# B&R Automation Studio project MotionTestBenchMaster (part 12)

```c
/*============================================================================*/
void mberror_client(tstMBT_SVars* inst, USINT clt)
/*----------------------------------------------------------------------------
  Function:

  History:

  Version | Date        | Author      | Description
  -----------------------------------------------------------------------------
     1.00 | 2010-okt-19 | H.Anderes    | creation
  ============================================================================*/
  {
  /* _LOCAL */
  STRING errstr[5+1];                        /* for status number */
  USINT  msize;                              /* for defensive programming, */
  /* _DYNAMIC */
  /*==========================================================================*/
  msize = sizeof(inst->cltInfo[clt].szMsg) - 1; /* http://www.manpagez.com/man/3/strncat/ */

  memset(inst->cltInfo[clt].szMsg, 0, sizeof(inst->cltInfo[clt].szMsg));
  switch (inst->uiStepCltHandler[clt])
  {
  /*-----------------------------------------------------------------------------
    DEBUG: client_handler state machine: W4_REQUEST
  ------------------------------------------------------------------------------*/
  case enMBTCP_CLT_HANDLER_W4_REQUEST:
    (void)strncat( inst->cltInfo[clt].szMsg,
                   "W4_REQUEST:",
                   msize - strlen(inst->cltInfo[clt].szMsg));
    (void)itoa(inst->stTcpSend[clt].status, (UDINT) &errstr);
    (void)strncat( inst->cltInfo[clt].szMsg,
                   errstr,
                   msize - strlen(inst->cltInfo[clt].szMsg));
    /* verfiy status */
    switch (inst->stTcpRecv[clt].status)
    {
    case ERR_OK:
      (void)strncat(inst->cltInfo[clt].szMsg, " status OK",
                    msize - strlen(inst->cltInfo[clt].szMsg));
      break;
    case ERR_FUB_BUSY:
      (void)strncat(inst->cltInfo[clt].szMsg, " FUB busy, trying again",
                    msize - strlen(inst->cltInfo[clt].szMsg));
      break;
    case tcpERR_NO_DATA:
      (void)strncat(inst->cltInfo[clt].szMsg, " Waiting (NO_DATA)",
                    msize - strlen(inst->cltInfo[clt].szMsg));
      break;
    case tcpERR_INVALID_IDENT:
    case tcpERR_NOT_CONNECTED:
      (void)strncat( inst->cltInfo[clt].szMsg,
                     " INVALID_IDENT, NOT_CONNECTED, disconnecting",
                     msize - strlen(inst->cltInfo[clt].szMsg));
      break;
    case tcpERR_SYSTEM:
      (void)strncat( inst->cltInfo[clt].szMsg,
                     " internal error while receiving",
                     msize - strlen(inst->cltInfo[clt].szMsg));
      /*************************************************************************/
      #ifdef _MBTCP_LOGGER_DEBUG
      ERRxwarning( mbtERR_NOT_CONNECTED,
                   inst->cltInfo[clt].udiIdent,
                   "MBTCP Server: TCP Recv tcpERR_SYSTEM");
      #endif
      /*************************************************************************/
      break;
    /*-------------------------------------------------------------------------*/
    case ERR_FUB_ENABLE_FALSE:
       (void)strncat(inst->cltInfo[clt].szMsg, " FUB not enabled",
                    msize - strlen(inst->cltInfo[clt].szMsg));
       break;
    /*-------------------------------------------------------------------------*/
    case tcpERR_NO_OOBDATA:
    case tcpERR_PARAMETER:
    case tcpERR_INVALID:
    default:
      (void)strncat(inst->cltInfo[clt].szMsg, " unknown error",
                    msize - strlen(inst->cltInfo[clt].szMsg));
      break;
    }
    break;
  /*-----------------------------------------------------------------------------
    DEBUG: client_handler state machine: SEND_RESPONSE
  ------------------------------------------------------------------------------*/
  case enMBTCP_CLT_HANDLER_SEND_RESPONSE:
    (void)strncat( inst->cltInfo[clt].szMsg,
                   "SEND_RESPONSE:",
                   msize - strlen(inst->cltInfo[clt].szMsg));
    (void)itoa(inst->stTcpSend[clt].status, (UDINT) &errstr);
    (void)strncat( inst->cltInfo[clt].szMsg,
                   errstr,
                   msize - strlen(inst->cltInfo[clt].szMsg));
    /* verify status */
    switch (inst->stTcpSend[clt].status)
    {
    case ERR_OK:
      (void)strncat(inst->cltInfo[clt].szMsg, " status OK",
                    msize - strlen(inst->cltInfo[clt].szMsg));
      break;
    case ERR_FUB_BUSY:
      (void)strncat(inst->cltInfo[clt].szMsg, " FUB busy, trying again",
                    msize - strlen(inst->cltInfo[clt].szMsg));
      break;
    case ERR_FUB_ENABLE_FALSE:
      (void)strncat(inst->cltInfo[clt].szMsg, " FUB not enabled",
                    msize - strlen(inst->cltInfo[clt].szMsg));
      break;
    case tcpERR_INVALID_IDENT:
      (void)strncat(inst->cltInfo[clt].szMsg, " ident not available",
                    msize - strlen(inst->cltInfo[clt].szMsg));
      break;
    case tcpERR_PARAMETER:
      (void)strncat(inst->cltInfo[clt].szMsg, " pData not set",
                    msize - strlen(inst->cltInfo[clt].szMsg));
      break;
    case tcpERR_SENTLEN:
      (void)strncat(inst->cltInfo[clt].szMsg,
                    " length of data to send <> specified length",
                    msize - strlen(inst->cltInfo[clt].szMsg));
      break;
    case tcpERR_WOULDBLOCK:
      (void)strncat(inst->cltInfo[clt].szMsg,
                    " data blocked out of socket's send buffer",
                    msize - strlen(inst->cltInfo[clt].szMsg));
      break;
    case tcpERR_NOT_CONNECTED:
      (void)strncat(inst->cltInfo[clt].szMsg,
                    " connection closed by opposite side",
                    msize - strlen(inst->cltInfo[clt].szMsg));
      break;
    case tcpERR_SYSTEM:
      (void)strncat(inst->cltInfo[clt].szMsg, " internal error while sending",
                    msize - strlen(inst->cltInfo[clt].szMsg));
      /************************************************************************/
      #ifdef _MBTCP_LOGGER_DEBUG
      ERRxwarning( mbtERR_NOT_CONNECTED,
                   inst->cltInfo[clt].udiIdent,
                   "MBTCP Server: Tcp Send tcpERR_SYSTEM");
      /************************************************************************/
      #endif
      break;
    default:
      (void)strncat(inst->cltInfo[clt].szMsg, " unknown error",
                    msize - strlen(inst->cltInfo[clt].szMsg));
      break;
    }
    break;
  /*-----------------------------------------------------------------------------
    DEBUG: client_handler state machine: DISCONNECT
  ------------------------------------------------------------------------------*/
  case enMBTCP_CLT_HANDLER_DISCONNECT:
    (void)strncat( inst->cltInfo[clt].szMsg,
                   "DISCONNECT:TCP_CLOSE:",
                   msize - strlen(inst->cltInfo[clt].szMsg));
    (void)itoa(inst->stTcpClose[clt].status, (UDINT) &errstr);
    (void)strncat( inst->cltInfo[clt].szMsg,
                   errstr,
                   msize - strlen(inst->cltInfo[clt].szMsg));
    /* verfiy status */
    switch (inst->stTcpClose[clt].status)
    {
    case ERR_OK:
      (void)strncat(inst->cltInfo[clt].szMsg, " OK. Client connection closed",
                    msize - strlen(inst->cltInfo[clt].szMsg));
      /************************************************************************/
      #ifdef _MBTCP_LOGGER_EVENT
      ERRxwarning( mbtEVENT_CLOSE_CLIENT,
                   inst->stTcpClose[clt].ident,
                   "MBTCP Server: Close Client");
      #endif
      /************************************************************************/
      break;
    case ERR_FUB_BUSY:
      (void)strncat(inst->cltInfo[clt].szMsg, " FUB_BUSY, Still trying...",
                    msize - strlen(inst->cltInfo[clt].szMsg));
      break;
    case tcpERR_INVALID_IDENT:
      (void)strncat(inst->cltInfo[clt].szMsg, " INVALID_IDENT",
                    msize - strlen(inst->cltInfo[clt].szMsg));
      break;
    case ERR_FUB_ENABLE_FALSE:
      (void)strncat(inst->cltInfo[clt].szMsg, " FUB_ENABLE_FALSE",
                    msize - strlen(inst->cltInfo[clt].szMsg));
      break;
    default:
      (void)strncat(inst->cltInfo[clt].szMsg, " unknown error",
                    msize - strlen(inst->cltInfo[clt].szMsg));
      break;
    }
    break;
  }
  /*==========================================================================*/
  } /* mberror */

/******************************************************************************
 * END OF CODE
 ******************************************************************************/
/*
Local Variables:
c-file-style: bsd
c-basic-offset: 2
comment-column: 45
End:
 */
```

#### MBTMaster.h
```c
/*****************************************************************************
 * Copyright:    B&R Industrie-Automation AG
 *
 * Project:      Library MBTCP
 *
 * Target:       B&R-PCC
 *
 * AR-Version:   B 2.01
 *
 * AS-Version:   V 3.0.71.16.SP01
 *
 * Filename:     MBTMaster.h
 *
 * Function:     module-description
 *
 * Dependencies: description of all dependencies
 *
 *****************************************************************************
 * History:
 *
 * Version | Date        | Author      | Description
 * --------------------------------------------------------------------------
 *    1.00 | 2008-Sep-30 | H.Anderes    | creation
 *****************************************************************************/

/*****************************************************************************
 * includes
 *****************************************************************************/
#ifndef MBTMASTER_H_
#define MBTMASTER_H_
/* ansi-c import */
#include <string.h>
/* system import */
#include <bur/plc.h>                         /* IEC data types */
#include <asstring.h>
#include <brsystem.h>
#include <astcp.h>
#include <convert.h>
#include <sys_lib.h>
/* user defined import */
#include "MBTCP.h"

/*#define _MBTCP_LOGGER_DEBUG*/    /* if defined, errors are logged into the logger */
/*#define _MBTCP_LOGGER_EVENT*/    /* if defined, events are logged into the logger */

#ifdef __i386__
#define SWAPUINT        swapUINT
#define SWAPINT         swapINT
#else
#define SWAPUINT
#define SWAPINT
#endif

/*****************************************************************************
 * constants / macros
 *****************************************************************************/
#define NELEMS(array)           (sizeof(array) / sizeof(array[0]))
/* Booleans, switches
 */
enum {
  FALSE                   = 0,
  TRUE                    = 1,
  EXIT_FAILURE            = 1,
  ON                      = 0xFF00,
  OFF                     = 0x0000
};

#define MAX_COILS    2000
#define MAX_REGISTER 127
/*****************************************************************************
 * type definitions
 *****************************************************************************/
/* STEP values
 */
enum {
  INIT                    = 0,
  WAIT_SERVER             = 5,
  OPEN_PORT               = 10,
  IOCTL                   = 15,
  WAIT_CONNECTION         = 20,
  WAIT_REQUEST            = 30,
  SEND_ANSWER             = 40,
  SEND_REQUEST            = 50,
  WAIT_ANSWER             = 60,
  CLOSE_PORT              = 70,
  FATAL_ERROR0            = 240,
  FATAL_ERROR1            = 241,
  FATAL_ERROR2            = 242,
  FATAL_ERROR3            = 243,
  FATAL_ERROR4            = 244,
  FATAL_ERROR5            = 245,
  FATAL_ERROR6            = 246,
  FATAL_ERROR7            = 247,
  FATAL_ERROR8            = 248,
  FATAL_ERROR9            = 249,
  FATAL_ERROR10           = 250,
  FATAL_ERROR             = 251,
  FINAL_ERROR			  = 252,

  DISABLE                 = 65534,
  BUSY                    = 65535
};

/* Modbus function codes
 */
enum {
  READ_COILS                            = 0x01,
  READ_DISCRETE_INPUTS                  = 0x02,
  READ_HOLDING_REGISTERS                = 0x03,
  READ_INPUT_REGISTERS                  = 0x04,
  WRITE_SINGLE_COIL                     = 0x05,
  WRITE_SINGLE_REGISTER                 = 0x06,
  WRITE_MULTIPLE_COILS                  = 0x0F,
  WRITE_MULTIPLE_REGISTERS              = 0x10,
  READ_WRITE_MULTIPLE_REGISTERS         = 0x17
};
/* Modbus protocol exception codes
 */
enum {
  MB_ILLEGAL_FUNCTION                   = 0x01,
  MB_ILLEGAL_DATA_ADDRESS               = 0x02,
  MB_ILLEGAL_DATA_VALUE                 = 0x03,
  MB_SLAVE_DEVICE_FAILURE               = 0x04,
  MB_ACKNOWLEDGE                        = 0x05,
  MB_SLAVE_DEVICE_BUSY                  = 0x06,
  MB_MEMORY_PARITY_ERROR                = 0x08,
  MB_GATEWAY_PATH_UNAVAILABLE           = 0x0A,
  MB_GATEWAY_TARGET_DEV_FAILED_RESPOND  = 0x0B
};
/* Dimensions
 */
enum {
  MBT_SLAVE_PORT        = 502,
  MAX_OPEN_RETRIES      = 3,
  RECV_TIMEOUT_DFLT     = 500,               /* default timeout */
  IPADDR_L              = 18,
  MAX_NBR_REQUESTS      = 5,                 /* was 20 */
  MAX_BUFFER_LEN        = 1200,/*128,*/
  MESS_LEN              = 100,               /* error message length */
};

/* Datatypes */
typedef struct MBTMasterActionParam_typ
{
  USINT usiFCode;
  USINT usiUnit;
  UINT  uiReadAddr;
  UINT  uiReadQty;
  UDINT puiReadVal;
  UINT  uiWriteAddr;
  UINT  uiWriteQty;
  UDINT puiWriteVal;
  UDINT udiTimer;
} MBTMasterActionParam_typ;

typedef struct MBTMasterActionEnable_typ
{
  BOOL bCyclic;
  BOOL bSingle;
} MBTMasterActionEnable_typ;

typedef struct tstMBT_MData
{
  MBTMasterActionEnable_typ actEnable[MAX_NBR_REQUESTS];
  MBTMasterActionParam_typ actParam[MAX_NBR_REQUESTS];
} tstMBT_MData;

typedef struct
{
  BOOL                  bEnable;
  STRING                slvIPAddr[IPADDR_L];
  UINT                  uiPort;
  UINT                  uiRecvTimeout;
  UDINT                 udiCycleTime;
  tstMBT_MData*         pData;
  UINT                  uiStep;
  TcpOpen_typ           stTcpOpen;
  TcpIoctl_typ          stTcpIoctl;
  TcpClient_typ         stTcpClient;
  TcpSend_typ           stTcpSend;
  TcpRecv_typ           stTcpRecv;
  TcpClose_typ          stTcpClose;
  USINT                 usiLastReq;
  UDINT                 udiRecvTimer;
  UDINT                 udiSendTimer[MAX_NBR_REQUESTS];
  USINT                 usiSendBuf[MAX_BUFFER_LEN];
  USINT                 usiRecvBuf[MAX_BUFFER_LEN];
  BOOL                  bRecvOK;
  UINT                  uiStatus;
  UINT                  uiTxID;
  UDINT                 udiWrongMsg;
  STRING                szMsg[MESS_LEN];
  tcpLINGER_typ         mLinger;
  USINT                 usiOpenRetries;
  USINT                 usiSendCnt;
} tstMBT_MVars;

/*****************************************************************************
 * functions protoytpes
 ****************************************************************************/
void  fMBTMStates(tstMBT_MVars* inst);
UINT create_request_to_server(tstMBT_MVars*   inst,
                               tstMBT_MData*   config,
                               USINT           usiOp,
                               USINT*          usiSendBuf,
                               UINT            uiTxID);
USINT analyze_answer_from_server(tstMBT_MVars* inst,
                                 tstMBT_MData* config,
                                 USINT         usiOp,
                                 USINT*        usiRecvBuf,
                                 UINT          uiTxID);

/****************************************************************************
 * END OF CODE
 ****************************************************************************/
/*
Local Variables:
c-file-style: bsd
c-basic-offset: 2
comment-column: 45
End:
 */
#endif /* MBTMASTER_H_ */
```

#### MBTMaster.c
```c
/******************************************************************************
 * Copyright:    B&R Industrie-Automation AG
 *
 * Project:      Library MBTCP
 *
 * Target:       B&R-PCC
 *
 * AR-Version:   B 2.01
 *
 * AS-Version:   V 3.0.71.16.SP01
 *
 * Filename:     MBTMaster.c
 *
 * Function:     module-description
 *
 * Dependencies: description of all dependencies
 *
 ******************************************************************************
 * History:
 *
 * Version | Date        | Author      | Description
 * ----------------------------------------------------------------------------
 *    1.00 | 2008-Sep-30 | H.Anderes   | creation
 *    2.00 | 2010-okt-04 | H.Anderes   | refactory
 *****************************************************************************/

/******************************************************************************
 * includes
 *****************************************************************************/
/* ansi-c import */
/* system import */
/* user defined import */
#include "MBTMaster.h"

/******************************************************************************
 * functions
 ******************************************************************************/
/*============================================================================*/
void fMBTMStates(tstMBT_MVars* inst)
/*----------------------------------------------------------------------------
  Function:

  History:

  Version | Date        | Author      | Description
  ----------------------------------------------------------------------------
  1.00    | 2008-sep-30 | H.Anderes    | creation
  2.00    | 2010-okt-04 | H.Anderes   | refactory
  ============================================================================*/
{
  /* _LOCAL */
  UINT uiFatalErrNum;
  USINT i, usiOp;                            /* usiOp: number of operations */
  USINT recv_status;
  /* _DYNAMIC */
  /*==========================================================================*/
  /* check if a null pointer is passed to the fub */
  if (inst == NULL)
  {
    return;
  }
  /*--------------------------------------------------------------------------------
    state machine : Modbus TCP Master
  ---------------------------------------------------------------------------------*/
  switch(inst->uiStep)
  {
  /*-----------------------------------------------------------------------------
    INIT: initialize TcpSend and TCPRecv
  ------------------------------------------------------------------------------*/
  case INIT:
    inst->stTcpSend.pData   = (UDINT)inst->usiSendBuf;
    inst->stTcpRecv.pData   = (UDINT)inst->usiRecvBuf;
    inst->stTcpRecv.datamax = MAX_BUFFER_LEN;
    inst->uiStep            = DISABLE;
    /* FALL THROUGH */
  /*-----------------------------------------------------------------------------
    DISBALE: waits until the fub is enabled
  ------------------------------------------------------------------------------*/
  case DISABLE:
    if(inst->bEnable)
    {
      inst->uiStep = OPEN_PORT;
    }
    break;
  /*-----------------------------------------------------------------------------
    OPEN: opens a TCP - socket
  ------------------------------------------------------------------------------*/
  case OPEN_PORT:
    inst->stTcpOpen.enable = 1;
    inst->stTcpOpen.port   = 0;
    /* call TcpOpen() */
    TcpOpen(&inst->stTcpOpen);
    /* verfiy status */
    switch (inst->stTcpOpen.status)
    {
    /*-------------------------------------------------------------------------*/
    case ERR_OK:
      inst->stTcpClient.enable     = 1;
      inst->stTcpClient.ident      = inst->stTcpOpen.ident;
      inst->stTcpClient.pServer    = (UDINT)inst->slvIPAddr;
      inst->stTcpClient.portserv   = inst->uiPort;
      inst->stTcpSend.ident        = inst->stTcpOpen.ident;
      inst->stTcpRecv.ident        = inst->stTcpOpen.ident;
      inst->uiStep                 = IOCTL;
      /************************************************************************/
      #ifdef _MBTCP_LOGGER_EVENT
	     ERRxwarning( mbtEVENT_OPEN_PORT,
                   inst->stTcpOpen.ident,
                   "MBTCP Client: Open Port");
      #endif
      /************************************************************************/
      break;
    /*-------------------------------------------------------------------------*/
    case ERR_FUB_BUSY:
      /* do nothing */
      break;
    /*-------------------------------------------------------------------------*/
    case tcpERR_NOMORE_IDENTS:
    case tcpERR_ALREADY_EXIST:
    case tcpERR_SOCKET_CREATE:
    case tcpERR_SOCKET_BIND:
    case tcpERR_INTERFACE:
    case tcpERR_SYSTEM:
    case ERR_FUB_ENABLE_FALSE:
    default:
      inst->uiStatus = inst->stTcpOpen.status;
      inst->uiStep   = FATAL_ERROR0;
      break;
    }
    break;
  /*-----------------------------------------------------------------------------
    IOCTRL: configuration of the TCP - connection
  ------------------------------------------------------------------------------*/
  case IOCTL:
    /* set linger that the connection is not abort immediately */
    inst->mLinger.lOnOff     = 0;
    inst->mLinger.lLinger    = 0;
     /* initialize fub */
    inst->stTcpIoctl.enable 	= 1;
    inst->stTcpIoctl.ident	  = inst->stTcpOpen.ident;
    inst->stTcpIoctl.ioctl 	 = tcpSO_LINGER_SET;
    inst->stTcpIoctl.pData	  = (UDINT)&inst->mLinger;
    inst->stTcpIoctl.datalen	= sizeof(tcpLINGER_typ);
    /* call  TcpIoctl()n */
    TcpIoctl(&inst->stTcpIoctl);
    /* verify status */
    switch (inst->stTcpIoctl.status)
    {
    /*-------------------------------------------------------------------------*/
    case ERR_OK:
      inst->usiOpenRetries = 0;      /* we reset prior to next step */
      inst->uiStep         = WAIT_CONNECTION;
      break;
    /*-------------------------------------------------------------------------*/
    case ERR_FUB_BUSY:
      inst->uiStep = IOCTL;
      break;
    /*-------------------------------------------------------------------------*/
    case tcpERR_INVALID_IDENT:
      inst->uiStatus = inst->stTcpIoctl.status;
      if (inst->usiOpenRetries < MAX_OPEN_RETRIES)
      {
        inst->uiStep = OPEN_PORT;
        inst->usiOpenRetries++;
        /************************************************************************/
        #ifdef _MBTCP_LOGGER_DEBUG
		      ERRxwarning( mbtERR_OPEN_RETRIES_IOC,
                     inst->stTcpOpen.ident,
                     "MBTCP Client: OPEN Retries IOCTL");
        #endif
        /************************************************************************/
      }
      else
      {
        inst->uiStep = FATAL_ERROR1;
      }
      break;
    /*-------------------------------------------------------------------------*/
    case tcpERR_PARAMETER:
      inst->uiStatus = inst->stTcpIoctl.status;
      inst->uiStep   = CLOSE_PORT;
      break;
    /*-------------------------------------------------------------------------*/
    case tcpERR_INVALID_IOCTL:
    case ERR_FUB_ENABLE_FALSE:
    default:
      inst->uiStatus = inst->stTcpIoctl.status;
      inst->uiStep   = FATAL_ERROR2;
      break;
    }
    break;
  /*-----------------------------------------------------------------------------
    WAIT: waits until a connection to a TCP Server is acc
  ------------------------------------------------------------------------------*/
  case WAIT_CONNECTION:
    inst->stTcpClient.enable = 1;
    /* call TcpClient() */
    TcpClient(&inst->stTcpClient);
    /* verify status */
    switch (inst->stTcpClient.status)
    {
    /*-------------------------------------------------------------------------*/
    case ERR_OK:
      inst->uiStep = SEND_REQUEST;
      break;
    /*-------------------------------------------------------------------------*/
    case ERR_FUB_BUSY:
      /* do nothing */
	     strcpy( inst->szMsg,
              "WAIT_CONNECTION:TcpClient: Wait Connection");
      break;
    /*-------------------------------------------------------------------------*/
    case tcpERR_INVALID:
   	  inst->uiStep = CLOSE_PORT;
      /*************************************************************************/
      #ifdef _MBTCP_LOGGER_DEBUG
   	  ERRxwarning( tcpERR_INVALID,
                   inst->stTcpClient.ident,
                   "MBTCP Client: Wait connecction; Invalid ");
      #endif
      /*************************************************************************/
      break;
    /*-------------------------------------------------------------------------*/
    case tcpERR_ALREADY_CONNECTED:
      inst->uiStep = CLOSE_PORT;
      /*************************************************************************/
      #ifdef _MBTCP_LOGGER_DEBUG
	     ERRxwarning( tcpERR_ALREADY_CONNECTED,
                             inst->stTcpClient.ident,
                             "MBTCP Client: Wait connecction; Already connected");
      #endif
      /*************************************************************************/
      break;
    /*-------------------------------------------------------------------------*/
    case tcpERR_SYSTEM:
    case ERR_FUB_ENABLE_FALSE:
    default:
      inst->uiStep = FATAL_ERROR3;
      break;
    }
    break;
  /*-----------------------------------------------------------------------------
    CREATE: creates the request
  ------------------------------------------------------------------------------*/
  case SEND_REQUEST:
    if (inst->bEnable)
    {
      inst->bRecvOK = FALSE;
      /* cycle through list of Modbus operations for MAX_NBR_REQUESTS times */
      for (i = inst->usiLastReq + 1;
           i < (MAX_NBR_REQUESTS + inst->usiLastReq + 1);
           i++)
      {
        usiOp = i % MAX_NBR_REQUESTS;
        if ((*(inst->pData)).actEnable[usiOp].bSingle)
        {
          inst->udiSendTimer[usiOp] =
            (*(inst->pData)).actParam[usiOp].udiTimer;
        }
        if ( (((*(inst->pData)).actEnable[usiOp].bCyclic)
              || ((*(inst->pData)).actEnable[usiOp].bSingle)))
        {
          if (inst->udiSendTimer[usiOp]
              >= (*(inst->pData)).actParam[usiOp].udiTimer)
          {
            inst->usiLastReq = usiOp;
            inst->uiStep = SEND_REQUEST + 1;
            inst->uiTxID++;
            inst->stTcpSend.datalen =
                create_request_to_server((tstMBT_MVars*)(inst),
                                       (tstMBT_MData*)(inst->pData),
                                       usiOp,
                                       inst->usiSendBuf,
                                       inst->uiTxID);
            inst->udiSendTimer[usiOp] = 0;
            break;
          }
          else
          {
            inst->udiSendTimer[usiOp] += inst->udiCycleTime;
          }
        }
        else
        {
          inst->udiSendTimer[usiOp]
            = (*(inst->pData)).actParam[usiOp].udiTimer;
        }
      }
    }
    else
    {
      inst->uiStep = CLOSE_PORT;
    }
    break;
  /*-----------------------------------------------------------------------------
    SEND: sends the created request to the server/slave
  ------------------------------------------------------------------------------*/
  case SEND_REQUEST + 1:
    if (inst->bEnable)
    {
      inst->stTcpSend.enable = 1;
      /* call TcpSend() */
      TcpSend(&inst->stTcpSend);
      /* verfiy status */
      switch (inst->stTcpSend.status)
      {
      /*-------------------------------------------------------------------------*/
      case ERR_OK:
        inst->usiSendCnt   = 0;
        inst->udiRecvTimer = 0;
        inst->uiStep       = WAIT_ANSWER;
        break;
      /*-------------------------------------------------------------------------*/
      case ERR_FUB_BUSY:
	       /* do nothing */
		      strcpy( inst->szMsg,
                "SEND_REQUEST + 1:TcpSend: ERR_FUB_BUSY");
	  	    break;
      /*-------------------------------------------------------------------------*/
      case tcpERR_WOULDBLOCK:
         /* send again */
         /************************************************************************/
         #ifdef _MBTCP_LOGGER_DEBUG
  	      ERRxwarning( tcpERR_WOULDBLOCK,
                      inst->stTcpClient.ident,
                      "MBTCP Client: Wouldblock");
         #endif
         /***********************************************************************/
   	   	break;
      /*-------------------------------------------------------------------------*/
      case tcpERR_SENTLEN:
        /* send length not ok. send again */
        /************************************************************************/
        #ifdef _MBTCP_LOGGER_DEBUG
        ERRxwarning( tcpERR_SENTLEN,
                     inst->stTcpClient.ident,
                     "MBTCP Client: Send lenght not Ok");
        #endif
        /************************************************************************/
        break;
      /*------------------------------------------------------------------------*/
      case tcpERR_NOT_CONNECTED:
        inst->uiStep = CLOSE_PORT;
        /************************************************************************/
        #ifdef _MBTCP_LOGGER_DEBUG
		      ERRxwarning( tcpERR_NOT_CONNECTED,
                     inst->stTcpClient.ident,
                     "MBTCP Client: Not connected");
        #endif
        /************************************************************************/
        break;
      /*-------------------------------------------------------------------------*/
      case tcpERR_INVALID_IDENT:
      case tcpERR_PARAMETER:
      case tcpERR_SYSTEM:
      default:
        inst->uiStep = FATAL_ERROR4;
        break;
      }
    }
    else
    {
      inst->uiStep = CLOSE_PORT;
    }
    break;
  /*-----------------------------------------------------------------------------
    WAIT: waits until a response is received or a timeout occured
  ------------------------------------------------------------------------------*/
  case WAIT_ANSWER:
    if (inst->bEnable)
    {
      inst->udiRecvTimer += inst->udiCycleTime;
      if (inst->udiRecvTimer >= inst->uiRecvTimeout)
      {
        /* send again after timeout */
        inst->uiStep = SEND_REQUEST;
        /************************************************************************/
        #ifdef _MBTCP_LOGGER_DEBUG
		      ERRxwarning( mbtERR_TIMEOUT,
                     inst->stTcpClient.ident,
                     "MBTCP Client: Receive Timeout");
        #endif
        /************************************************************************/
        break;
      }
      inst->stTcpRecv.enable = 1;
      /* call TcpRecv() */
      TcpRecv(&(inst->stTcpRecv));
      /* verfiy status */
      switch (inst->stTcpRecv.status)
      {
      /*-------------------------------------------------------------------------*/
      case ERR_OK:
        if (inst->stTcpRecv.recvlen > 8)
        {
          recv_status =
            analyze_answer_from_server((tstMBT_MVars*)(inst),
                                       (tstMBT_MData*)(inst->pData),
                                       inst->usiLastReq,
                                       inst->usiRecvBuf,
                                       inst->uiTxID);
        }
        else
        {
          recv_status = 1;
        }
        if(recv_status)
		      {
           inst->udiWrongMsg++;
           /**********************************************************************/
           #ifdef _MBTCP_LOGGER_DEBUG
 		        ERRxwarning( mbtERR_RESPONSE,
                        inst->stTcpRecv.ident,
                        "MBTCP Client: Response not Ok");
           #endif
           /**********************************************************************/

        }
        else
        {
          (*(inst->pData)).actEnable[inst->usiLastReq].bSingle = 0;
        }
        inst->uiStep = SEND_REQUEST;
        break;
      /*-------------------------------------------------------------------------*/
      case ERR_FUB_BUSY:
      case ERR_FUB_ENABLE_FALSE:
      case tcpERR_NO_DATA:
        /* do nothing */
		      strcpy(inst->szMsg, "WAIT_ANSWER:TcpClient: tcpERR_NO_DATA");
        break;
      /*-------------------------------------------------------------------------*/
      case tcpERR_NOT_CONNECTED:
        inst->uiStep = SEND_REQUEST;
		      strcpy(inst->szMsg, "WAIT_ANSWER:TcpClient: tcpERR_NOT_CONNECTED");
        break;
      /*-------------------------------------------------------------------------*/
      case tcpERR_INVALID_IDENT:
      case tcpERR_PARAMETER:
      case tcpERR_INVALID:
      case tcpERR_NO_OOBDATA:
      case tcpERR_SYSTEM:
      default:
        inst->uiStep = FATAL_ERROR5;
        break;
      }
    }
    else
    {
      inst->uiStep = CLOSE_PORT;
    }
    break;
  /*-----------------------------------------------------------------------------
    CLOSE: closes the TCP - Socket
  ------------------------------------------------------------------------------*/
  case CLOSE_PORT:
    inst->stTcpClose.enable = 1;
    inst->stTcpClose.ident  = inst->stTcpOpen.ident;
    /*
      inst->stTcpClose.how    = tcpSHUT_RD | tcpSHUT_WR;
    */
    inst->stTcpClose.how    = 0;
    /* call TcpClose() */
    TcpClose(&inst->stTcpClose);
    /* verfiy status */
    switch (inst->stTcpClose.status)
    {
    /*-------------------------------------------------------------------------*/
    case ERR_OK:
      inst->uiStep = DISABLE;
      /*************************************************************************/
      #ifdef _MBTCP_LOGGER_DEBUG
	     ERRxwarning( mbtEVENT_CLOSE_PORT,
                   inst->stTcpClose.ident,
                   "MBTCP Client: Close Port");
      #endif
      /*************************************************************************/
      break;
    /*-------------------------------------------------------------------------*/
    case ERR_FUB_BUSY:
      /* do nothing */
      break;
    /*-------------------------------------------------------------------------*/
    case tcpERR_INVALID_IDENT:
      inst->uiStep = WAIT_CONNECTION;
      break;
    /*-------------------------------------------------------------------------*/
    case ERR_FUB_ENABLE_FALSE:
    default:
      inst->uiStep = FATAL_ERROR6;
      break;
    }
    break;
  /*-----------------------------------------------------------------------------
    FATAL ERROR: a fatal error occured
  ------------------------------------------------------------------------------*/
  case FATAL_ERROR0:
  case FATAL_ERROR1:
  case FATAL_ERROR2:
  case FATAL_ERROR3:
  case FATAL_ERROR4:
  case FATAL_ERROR5:
  case FATAL_ERROR6:
  default:
   /* vefiy in which state the fatal error occured */
  	switch(inst->uiStep)
	  {
	  case FATAL_ERROR0: uiFatalErrNum = 0; break;
  	case FATAL_ERROR1: uiFatalErrNum = 1; break;
  	case FATAL_ERROR2: uiFatalErrNum = 2; break;
  	case FATAL_ERROR3: uiFatalErrNum = 3; break;
  	case FATAL_ERROR4: uiFatalErrNum = 4; break;
  	case FATAL_ERROR5: uiFatalErrNum = 5; break;
  	case FATAL_ERROR6: uiFatalErrNum = 6; break;
	  default:
		   uiFatalErrNum = 7; break;
	  }
	   /*************************************************************************/
    #ifdef _MBTCP_LOGGER_DEBUG
   	ERRxwarning( mbtERR_FATAL_ERROR,
                 uiFatalErrNum,
                 "MBTCP Client: FATAL ERROR State Machine");
    #endif
    /*************************************************************************/
   	inst->uiStep = FINAL_ERROR;
    break;

  case FINAL_ERROR:
  	/*Do nothing until Reboot RPS*/
  	break;
  }
}

/*============================================================================*/
UINT create_request_to_server(tstMBT_MVars* inst,
                               tstMBT_MData* config,
                               USINT         usiOp,
                               USINT*        usiSendBuf,
                               UINT          uiTxID)
/*----------------------------------------------------------------------------
  Function:

  History:

  Version | Date        | Author      | Description
  ----------------------------------------------------------------------------
     1.00 | 2008-sep-30 | H.Anderes    | creation
  ============================================================================*/
{
  UINT  uint_var, data_len, i;
  INT  int_var;
  UINT  value;
  UINT  val;
 /*==========================================================================*/
  data_len = 0;

  memset(usiSendBuf, 0, MAX_BUFFER_LEN);
  /* Transaction id: 2 bytes */
  uint_var = SWAPUINT(uiTxID);
  memmove(&usiSendBuf[0], &uint_var, sizeof(uint_var));
  /* Protocol id: 2 bytes */
  uint_var = 0;
  memmove(&usiSendBuf[2], &uint_var, sizeof(uint_var));
  /* Length: 2 bytes */
  /* Unit: 1 byte */
  usiSendBuf[6] = (*config).actParam[usiOp].usiUnit;

  switch((*config).actParam[usiOp].usiFCode)
  {
  /*-------------------------------------------------------------------------
      READ: read coils
  --------------------------------------------------------------------------*/
  case READ_COILS:
    /* Function code: 1 byte */
    usiSendBuf[7] = READ_COILS;
    /* Starting address: 2 bytes */
    uint_var = SWAPUINT((*config).actParam[usiOp].uiReadAddr);
    memmove(&usiSendBuf[8], &uint_var, sizeof(uint_var));
    /* Coils number: 2 bytes */
    uint_var = SWAPUINT((*config).actParam[usiOp].uiReadQty);
    memmove(&usiSendBuf[10], &uint_var, sizeof(uint_var));
    /* Data len */
    data_len = 6;
    inst->bRecvOK = FALSE;
    break;
  /*-------------------------------------------------------------------------
      READ: read discrete inputs
  --------------------------------------------------------------------------*/
  case READ_DISCRETE_INPUTS:
    /* Function code: 1 byte */
    usiSendBuf[7] = READ_DISCRETE_INPUTS;
    /* Starting address: 2 bytes */
    uint_var = SWAPUINT((*config).actParam[usiOp].uiReadAddr);
    memmove(&usiSendBuf[8], &uint_var, sizeof(uint_var));
    /* Inputs number: 2 bytes */
    uint_var = SWAPUINT((*config).actParam[usiOp].uiReadQty);
    memmove(&usiSendBuf[10], &uint_var, sizeof(uint_var));
    /* Data len */
    data_len = 6;
    inst->bRecvOK = FALSE;
    break;
  /*-------------------------------------------------------------------------
      READ: read holding registers
  --------------------------------------------------------------------------*/
  case READ_HOLDING_REGISTERS:
    /* Function code: 1 byte */
    usiSendBuf[7] = READ_HOLDING_REGISTERS;
    /* Starting address: 2 bytes */
    uint_var = SWAPUINT((*config).actParam[usiOp].uiReadAddr);
    memmove(&usiSendBuf[8], &uint_var, sizeof(uint_var));
    /* Holding registers number: 2 bytes */
    uint_var = SWAPUINT((*config).actParam[usiOp].uiReadQty);
    memmove(&usiSendBuf[10], &uint_var, sizeof(uint_var));
    /* Data len */
    data_len = 6;
    inst->bRecvOK = FALSE;
    break;
  /*-------------------------------------------------------------------------
      READ: read input registers
  --------------------------------------------------------------------------*/
  case READ_INPUT_REGISTERS:
    /* Function code: 1 byte */
    usiSendBuf[7] = READ_INPUT_REGISTERS;
    /* Starting address: 2 bytes */
    uint_var = SWAPUINT((*config).actParam[usiOp].uiReadAddr);
    memmove(&usiSendBuf[8], &uint_var, sizeof(uint_var));
    /* Input registers number: 2 bytes */
    uint_var = SWAPUINT((*config).actParam[usiOp].uiReadQty);
    memmove(&usiSendBuf[10], &uint_var, sizeof(uint_var));
    /* Data len */
    data_len = 6;
    inst->bRecvOK = FALSE;
    break;
  /*-------------------------------------------------------------------------
      WRITE: write single coil
  --------------------------------------------------------------------------*/
  case WRITE_SINGLE_COIL:
    /* Function code: 1 byte */
    usiSendBuf[7] = WRITE_SINGLE_COIL;
    /* Starting address: 2 bytes */
    uint_var = SWAPUINT((*config).actParam[usiOp].uiWriteAddr);
    memmove(&usiSendBuf[8], &uint_var, sizeof(uint_var));
    /* Value: 2 bytes */
    memmove(&val, (UINT *)((*config).actParam[usiOp].puiWriteVal), sizeof(UINT));
    if ((BOOL)(val))
      value = ON;
    else
      value = OFF;
    int_var = SWAPUINT(value);
    memmove(&usiSendBuf[10], &int_var, sizeof(int_var));
    /* Data len */
    data_len = 6;
    inst->bRecvOK = FALSE;
    break;
  /*-------------------------------------------------------------------------
      WRITE: write single register
  --------------------------------------------------------------------------*/
  case WRITE_SINGLE_REGISTER:
    /* Function code: 1 byte */
    usiSendBuf[7] = WRITE_SINGLE_REGISTER;
    /* Starting address: 2 bytes */
    uint_var = SWAPUINT((*config).actParam[usiOp].uiWriteAddr);
    memmove(&usiSendBuf[8], &uint_var, sizeof(uint_var));
    /* Value: 2 bytes */
    memmove(&val, (UINT *)(*config).actParam[usiOp].puiWriteVal, sizeof(UINT));
    value = (UINT)(val);
    uint_var = SWAPUINT(value);
    memmove(&usiSendBuf[10], &uint_var, sizeof(uint_var));
    /* Data len */
    data_len = 6;
    inst->bRecvOK = FALSE;
    break;
  /*-------------------------------------------------------------------------
      WRITE: write multiple coils
  --------------------------------------------------------------------------*/
  case WRITE_MULTIPLE_COILS:
    /* Function code: 1 byte */
    usiSendBuf[7] = WRITE_MULTIPLE_COILS;
    /* Starting address: 2 bytes */
    uint_var = SWAPUINT((*config).actParam[usiOp].uiWriteAddr);
    memmove(&usiSendBuf[8], &uint_var, sizeof(uint_var));
    /* Quantity: 2 bytes */
    uint_var = SWAPUINT((*config).actParam[usiOp].uiWriteQty);
    memmove(&usiSendBuf[10], &uint_var, sizeof(uint_var));
    /* Byte count: 1 byte */
    /* Number of usiSendBuf bytes needed to contain data */
    /* less than 8 binary digits: 1 byte */
    if ( (*config).actParam[usiOp].uiWriteQty % 8)
      usiSendBuf[12] = ((*config).actParam[usiOp].uiWriteQty / 8) + 1;
    else      /* more than 8 binary digits: quantity / 8 bytes */
      usiSendBuf[12] = (*config).actParam[usiOp].uiWriteQty / 8;
    /* Coil value: x byte */
    for (i = 0; i < (*config).actParam[usiOp].uiWriteQty; i++)
    {
      memmove(&val,
              (UINT *)((*config).actParam[usiOp].puiWriteVal  +  i * sizeof(UINT)),
              sizeof(UINT));
      if ((BOOL)(val))
        usiSendBuf[13 + (i/8)]
          = usiSendBuf[13 + (i/8)] | (USINT)(0x01 << (i%8));
      else
        usiSendBuf[13 + (i/8)]
          = usiSendBuf[13 + (i/8)] & (USINT)~(0x01 << (i%8));
    }
    /* Data len */
    data_len = 7 + usiSendBuf[12];
    inst->bRecvOK = FALSE;
    break;
  /*-------------------------------------------------------------------------
      WRITE: write multiple registers
  --------------------------------------------------------------------------*/
  case WRITE_MULTIPLE_REGISTERS:
    /* Function code: 1 byte */
    usiSendBuf[7] = WRITE_MULTIPLE_REGISTERS;
    /* Starting address: 2 bytes */
    uint_var = SWAPUINT((*config).actParam[usiOp].uiWriteAddr);
    memmove(&usiSendBuf[8], &uint_var, sizeof(uint_var));
    /* Quantity: 2 bytes */
    uint_var = SWAPUINT((*config).actParam[usiOp].uiWriteQty);
    memmove(&usiSendBuf[10], &uint_var, sizeof(uint_var));
    /* Byte count: 1 byte */
    usiSendBuf[12] = (*config).actParam[usiOp].uiWriteQty * 2;
    /* Coil value: x byte */
    for(i = 0; i < (*config).actParam[usiOp].uiWriteQty; i++)
    {
      value = ((INT*)((*config).actParam[usiOp].puiWriteVal))[i];
      int_var = SWAPINT(value);
      memmove(&usiSendBuf[13 + (i*2)], &int_var, sizeof(int_var));
    }
    /* Data len */
    data_len = 7 + usiSendBuf[12];
    inst->bRecvOK = FALSE;
    break;
  /*-------------------------------------------------------------------------
     READ WRITE:read  write multiple registers
  --------------------------------------------------------------------------*/
  case READ_WRITE_MULTIPLE_REGISTERS:
    /* Function code: 1 byte */
    usiSendBuf[7] = READ_WRITE_MULTIPLE_REGISTERS;
    /* Read starting address: 2 bytes */
    uint_var = SWAPUINT((*config).actParam[usiOp].uiReadAddr);
    memmove(&usiSendBuf[8], &uint_var, sizeof(uint_var));
    /* Read quantity: 2 bytes */
    uint_var = SWAPUINT((*config).actParam[usiOp].uiReadQty);
    memmove(&usiSendBuf[10], &uint_var, sizeof(uint_var));
    /* Write starting address: 2 bytes */
    uint_var = SWAPUINT((*config).actParam[usiOp].uiWriteAddr);
    memmove(&usiSendBuf[12], &uint_var, sizeof(uint_var));
    /* write quantity: 2 bytes */
    uint_var = SWAPUINT((*config).actParam[usiOp].uiWriteQty);
    memmove(&usiSendBuf[14], &uint_var, sizeof(uint_var));
    /* Byte count: 1 byte */
    usiSendBuf[16] = (*config).actParam[usiOp].uiWriteQty * 2;
    /* Coil value: x byte */
    for(i = 0; i < (*config).actParam[usiOp].uiWriteQty; i++)
    {
      value = ((INT*)((*config).actParam[usiOp].puiWriteVal))[i];
      int_var = SWAPINT(value);
      memmove(&usiSendBuf[17 + (i*2)], &int_var, sizeof(int_var));
    }
    /* Data len */
    data_len = 11 + usiSendBuf[16];
    inst->bRecvOK = FALSE;
    break;
  default:
    break;
  }
  /* Length: 2 bytes */
  uint_var = SWAPUINT(data_len);
  memmove(&usiSendBuf[4], &uint_var, sizeof(uint_var));

  return (6 + data_len);
}

 /*==========================================================================*/
USINT analyze_answer_from_server(tstMBT_MVars* inst,
                                 tstMBT_MData* config,
                                 USINT         usiOp,
                                 USINT*        usiRecvBuf,
                                 UINT          uiTxID)
/*----------------------------------------------------------------------------
  Function:

  History:

  Version | Date        | Author      | Description
  ----------------------------------------------------------------------------
     1.00 | 2008-sep-30 | H.Anderes   | creation
     2.00 | 2010-okt-04 | H.Anderes   | refactory
  ============================================================================*/
{
  INT   int_var;
  UINT  uint_var, recv_tr_id, protocol_id, length, uiQty,i;
  USINT unit, function_code;
  UINT  coil_val, di_val;         /* was UDINT */
  /*==========================================================================*/

  coil_val = 0;
  di_val   = 0;
  /* (byte 0,1)  transition is */
  memmove(&uint_var, &(usiRecvBuf[0]), sizeof(uint_var));
  recv_tr_id = SWAPUINT(uint_var);
  /* (byte 2,3)  protocol id */
  memmove(&uint_var, &(usiRecvBuf[2]), sizeof(uint_var));
  protocol_id = SWAPUINT(uint_var);
  /* (byte 4,5)  length */
  memmove(&uint_var, &(usiRecvBuf[4]), sizeof(uint_var));
  length = SWAPUINT(uint_var);
  /* (byte 4,5)  length */
  unit = usiRecvBuf[6];
  /* (byte 7 ) function code */
  function_code = usiRecvBuf[7];

  if (    (recv_tr_id == uiTxID)
       && (protocol_id == 0)
       && (length > 0)
       && (function_code  < 0x80) )
  {

    switch(function_code)
    {
    /*-------------------------------------------------------------------------
      READ: read coils
    --------------------------------------------------------------------------*/
    case READ_COILS:
      /* Quantity: 1 byte */
      uiQty = usiRecvBuf[8];
      if (uiQty > MAX_COILS)
      {
        uiQty = MAX_COILS;
      }
      /* Coil value: x bytes */
      /* uiQty is number of bytes received */
      for (i = 0;(i < uiQty*8) && (i < (*config).actParam[usiOp].uiReadQty); i++) {
        coil_val = (UINT)(usiRecvBuf[9 + (i/8)] & (USINT)(0x01 << (i%8)));
        if ((BOOL)(coil_val))
          ((INT*)((*config).actParam[usiOp].puiReadVal))[i] = 1;
        else
          ((INT*)((*config).actParam[usiOp].puiReadVal))[i] = 0;
      }
      inst->bRecvOK = TRUE;
      break;
    /*-------------------------------------------------------------------------
      READ: read discrete inputs
    --------------------------------------------------------------------------*/
    case READ_DISCRETE_INPUTS:
      /* Quantity: 1 byte */
      uiQty = usiRecvBuf[8];
      if (uiQty > MAX_COILS)
      {
        uiQty = MAX_COILS;
      }
      /* Coil value: x byte */
      /* quantity is number of bytes received */
      for(i = 0; (i < uiQty*8) && (i < (*config).actParam[usiOp].uiReadQty); i++) {
        di_val = (UINT)(usiRecvBuf[9 + (i/8)] & (USINT)(0x01 << (i%8)));
         if ((BOOL)(di_val))
           ((INT*)((*config).actParam[usiOp].puiReadVal))[i] = 1;
         else
           ((INT*)((*config).actParam[usiOp].puiReadVal))[i] = 0;
      }
      inst->bRecvOK = TRUE;
      break;
    /*-------------------------------------------------------------------------
      READ: read hoding registers
    --------------------------------------------------------------------------*/
    case READ_HOLDING_REGISTERS:
      /* Quantity: 1 byte */
       uiQty = usiRecvBuf[8] / 2;
       if (uiQty > MAX_REGISTER)
       {
         uiQty = MAX_REGISTER;
       }
      /* Coil value: x byte */
      for(i = 0; i < uiQty; i++) {
        memmove(&int_var, &usiRecvBuf[9 + (i*2)], sizeof(int_var));
        ((INT*)((*config).actParam[usiOp].puiReadVal))[i] = SWAPINT(int_var);
      }
      inst->bRecvOK = TRUE;
      break;
    /*-------------------------------------------------------------------------
      READ: read input registers
    --------------------------------------------------------------------------*/
    case READ_INPUT_REGISTERS:
      /* Quantity: 1 byte */
      uiQty = usiRecvBuf[8] / 2;
      if (uiQty > MAX_REGISTER)
      {
        uiQty = MAX_REGISTER;
      }
      /* Coil value: x byte */
      for(i = 0; i < uiQty; i++) {
        memmove(&int_var, &usiRecvBuf[9 + (i*2)], sizeof(int_var));
        ((INT*)((*config).actParam[usiOp].puiReadVal))[i] = SWAPINT(int_var);
      }
      inst->bRecvOK = TRUE;
      break;
    /*-------------------------------------------------------------------------
      READ: read write multiple registers
    --------------------------------------------------------------------------*/
    case READ_WRITE_MULTIPLE_REGISTERS:
      /* Quantity: 1 byte */
      uiQty = usiRecvBuf[8] / 2;
      if (uiQty > MAX_REGISTER)
      {
        uiQty = MAX_REGISTER;
      }
      /* Coil value: x byte */
      for(i = 0; i < uiQty; i++) {
        memmove(&int_var, &usiRecvBuf[9 + (i*2)], sizeof(int_var));
        ((INT*)((*config).actParam[usiOp].puiReadVal))[i] = SWAPINT(int_var);
      }
      inst->bRecvOK = TRUE;
      break;

    default:
      inst->bRecvOK = TRUE;
      break;
    }
  }
  else
  { /* if (    (recv_tr_id == uiTxID)
            && (protocol_id == 0)
            && (length > 0)
            && (function_code  < 0x80) ) */
    /*************************************************************************/
    #ifdef _MBTCP_LOGGER_DEBUG
    if(protocol_id != 0)
    {
		    ERRxwarning( mbtERR_PROTOCOL_ID,
                   inst->stTcpRecv.ident,
                   "MBTCP Client: Protocol ID != 0");
    }
	   if(length == 0)
    {
		    ERRxwarning( mbtERR_RESPONSE,
                   inst->stTcpRecv.ident,
                   "MBTCP Client: Response lenght == 0");
    }
	   if(function_code  > 0x80)
    {
		    ERRxwarning( mbtERR_RESPONSE,
                    inst->stTcpRecv.ident,
                    "MBTCP Client: function_code  > 0x80");
    }
    #endif
    /*************************************************************************/

    return EXIT_FAILURE;
  }

  return ERR_OK;
}

/******************************************************************************
 * END OF CODE
 ******************************************************************************/
/*
Local Variables:
c-file-style: bsd
c-basic-offset: 2
comment-column: 45
End:
*/
```

#### Convert.c
```c
/******************************************************************************
 * Copyright:    B&R Industrie-Automation AG
 *
 * Project:      Library MBTCP
 *
 * Target:       B&R-PCC
 *
 * Filename:     Convert.c
 *
 * Function:     module-description
 *
 * Dependencies: description of all dependencies
 *
 ******************************************************************************
 * History:
 *
 * Version | Date        | Author       | Description
 * ----------------------------------------------------------------------------
 *    1.00 | 2012-aug-03 | H.Anderes    | creation
 *****************************************************************************/

/*****************************************************************************
 * includes
 *****************************************************************************/
/* ansi-c import */
/* system import */
#include <bur/plctypes.h>
/* user defined import */
#include "Convert.h"

INT swapINT (INT wInputValue)
{
 return (wInputValue << 8) + (USINT)(wInputValue >> 8);
}

UINT swapUINT (UINT wInputValue)
{
 return (wInputValue << 8) + (USINT)(wInputValue >> 8);
}

/*****************************************************************************
 * END OF CODE
 *****************************************************************************/
```

#### Convert.h
```c
/*****************************************************************************
 * Copyright:    B&R Industrie-Automation AG
 *
 * Project:      Library MBTCP
 *
 * Target:       B&R-PCC
 *
 * Filename:     Convert.h
 *
 * Function:     module-description
 *
 * Dependencies: description of all dependencies
 *
 *****************************************************************************
 * History:
 *
 * Version | Date        | Author      | Description
 * --------------------------------------------------------------------------
 *    1.00 | 2008-sep-19 | H.Anderes    | creation
 *****************************************************************************/

/*****************************************************************************
 * includes
 *****************************************************************************/
#ifndef CONVERT_H_
#define CONVERT_H_

#include <bur/plctypes.h>

INT swapINT (INT wInputValue);
UINT swapUINT (UINT wInputValue);

#endif /* CONVERT_H_ */
/*****************************************************************************
 * END OF CODE
 *****************************************************************************/
```

### Library Logical/00_AID/Libraries/Sidel_Libraries/ITC/TCP_COM (IEC, version 4.00.0)

#### TCP_COM.fun - Exported functions and function blocks
```iecst
(********************************************************************
 * COPYRIGHT --
 ********************************************************************
 * Package: TCP
 * File: TCP.typ
 * Author: Marco.Nicoli
 * Created: October 25, 2016 : Initial version
 *********************************************************************)

FUNCTION_BLOCK TCP_COM (*TCP communication function*)
	VAR_INPUT
		Enable_Com : BOOL; (*Enable Communication*)
		Enable_Server : BOOL; (*Enable the server mode (False = Client mode | True = Serve mode)*)
		ETH_Card : STRING[16] := 'IF2'; (*Optional Parameter
Work with the following syntax when using IF2 on board:
IF2
Work with the following syntax when using a POWERLINK card:
SL<x>.SS<y>.IF<z>.PLKETH or SL<x>.SS<y>.IF<z>.ETH
*)
		IP_Address : STRING[16]; (*Partner IP address. (e.g. '10.1.92.20') (as a string)*)
		Local_Port : UINT; (*Local port number.*)
		Remote_Port : UINT; (*Remote port number.*)
		Recv_Buffer : UDINT; (*Received data buffer address (string given as a pointer)*)
		Recv_Length : UDINT; (*Reiceved data maximum length (in bytes)*)
		Send_Buffer : UDINT; (*Data to send buffer address (string given as a pointer)*)
		Send_Length : UDINT; (*Sent data length (in bytes)*)
		Send_Time_Act : TIME; (*Data send time cadence (in ms) (typical value: 100ms)*)
		Rcv_Time_Out : TIME; (*Reception time out setpoint (in ms) (typical value: 1000ms)*)
	END_VAR
	VAR_OUTPUT
		Connection_OK : BOOL; (*True = both PLCs are connected*)
		PING_OK : BOOL;
		ERROR : BOOL;
		ERR_NO_RESPONSE : BOOL;
		ERR_INTERNAL : BOOL;
	END_VAR
	VAR
		WhoIsConnected : STRING[16]; (*Connected client IP address*)
		IP_AdressLocal : STRING[16];
		TON_SendTime : TON;
		TON_RcvTimeOut : TON;
		TON_TCP_EnDelay : TON;
		TON_ConnectionTimeOut : TON;
		ConnectionAttempt : UINT;
		fb_Ping : PING_Fun;
		fb_TcpOpen : TcpOpen; (*Communication opening function block*)
		fb_TcpServer : TcpServer; (*Server creation function block*)
		fb_TcpClient : TcpClient; (*Client function block*)
		fb_TcpSend : TcpSend; (*Data sending function block*)
		fb_TcpRecv : TcpRecv; (*Data receiving function block*)
		fb_TcpClose : TcpClose; (*Communication closing function block*)
		fb_CfgGetIPAddr : CfgGetIPAddr;
		oldTCP_Status : TCP_Status_Type;
		oldTCP_CommStatus : TCP_SendRec_Type;
		IP_LocalValid : BOOL;
		readResponse : BOOL;
		commResponse : BOOL;
		TCP_Status : TCP_Status_Type; (*Implemented communication block status*)
		TCP_CommStatus : TCP_SendRec_Type; (*Implemented communication block status*)
		TON_Connection_OK : TON;
	END_VAR
END_FUNCTION_BLOCK

FUNCTION_BLOCK PING_Fun (*TODO: Add your comment here*) (*$GROUP=User,$CAT=User,$GROUPICON=User.png,$CATICON=User.png*)
	VAR_INPUT
		enable : BOOL;
		IP_Address : STRING[80];
	END_VAR
	VAR_OUTPUT
		PING_OK : BOOL;
		ERROR : BOOL;
		ERR_NO_RESPONSE : BOOL;
		ERR_INTERNAL : BOOL;
	END_VAR
	VAR
		Status : Ping_Status_Type;
		Fb_IcmpPing : IcmpPing;
		PachetRecived : USINT;
		PachetSent : USINT;
		PachetLoss : USINT;
		readResponse : BOOL;
	END_VAR
END_FUNCTION_BLOCK
```

#### TCP_COM.typ - Exported data types
```iecst
(********************************************************************
 * COPYRIGHT --
 ********************************************************************
 * Package: TCP
 * File: TCP.typ
 * Author: Marco.Nicoli
 * Created: October 25, 2016 : Initial version
 *********************************************************************)

TYPE
	TCP_DataType : 	STRUCT
		Connection_OK : BOOL;
		Com_Status : UINT; (*(0=Connect OK;1=Not Enabled;2=Error Sending;3=Error Receiving;10=Connection Waiting)*)
		Recv_Buffer : ARRAY[0..20]OF USINT;
		Send_Buffer : ARRAY[0..20]OF USINT;
	END_STRUCT;
	TCP_Status_Type :
		(
		DISABLED,
		INITIALIZE_FB,
		INITIAL_PING,
		READ_LOCAL_IP,
		OPEN_TCP,
		CFG_SERVER,
		CFG_CLIENT,
		ESTABLISHED_CONNECTION_AS_SERVER,
		ESTABLISHED_CONNECTION_AS_CLIENT,
		CLOSE1,
		CLOSE2,
		RECONNECTION
		);
	TCP_SendRec_Type :
		(
		COMM_IDLE,
		SEND_DATA,
		RECEIVE_DATA,
		COMM_PING
		);
	Ping_Status_Type :
		(
		NO_EXECUTION,
		EXECUTION,
		SUCCESSFUL,
		NO_RESPONSE,
		ERROR_INTERNAL
		);
END_TYPE
```

#### TCP_COM.var - Exported constants
```iecst
(********************************************************************
 * COPYRIGHT --
 ********************************************************************
 * Library: TCP_COMM
 * File: TCP_COMM.var
 * Author: SIDEL Conveying France
 * Created: October 02, 2008
 ********************************************************************
 * Constants of library TCP_COM
 ********************************************************************)
VAR CONSTANT
	TCP_Connected_OK : USINT := 0;
	TCP_Error_Sending : USINT := 2;
	TCP_Connection_Waiting : USINT := 10;
	TCP_Error_Receiving : USINT := 3;
	TCP_Not_Enabled : UINT := 1;
END_VAR
```

#### TCP_Fun.st
```iecst
(********************************************************************
 * COPYRIGHT --
 ********************************************************************
 * Package: TCP
 * File: TCP.st
 * Author: Marco.Nicolì
 * Created: October 25, 2016 : Initial version
 * Modified: November 15, 2016 : Something
 ********************************************************************)

FUNCTION_BLOCK TCP_COM
	CASE TCP_Status OF
		DISABLED:
			ConnectionAttempt 	:= 0;
			PING_OK 			:= FALSE;
			ERR_INTERNAL		:= FALSE;
			ERR_NO_RESPONSE		:= FALSE;
			TON_TCP_EnDelay.IN 	:= Enable_Com;
			TON_TCP_EnDelay.PT 	:= t#2s;
			TON_TCP_EnDelay();
			IF TON_TCP_EnDelay.Q THEN
				TON_TCP_EnDelay(IN := FALSE);
				TCP_Status := INITIALIZE_FB;
			END_IF

		INITIALIZE_FB:
			fb_Ping.enable 		:= FALSE;
			fb_TcpOpen.enable	:= FALSE;
			fb_TcpServer.enable	:= FALSE;
			fb_TcpClient.enable	:= FALSE;
			fb_TcpSend.enable	:= FALSE;
			fb_TcpRecv.enable	:= FALSE;
			fb_TcpClose.enable	:= FALSE;
			fb_CfgGetIPAddr.enable := FALSE;
			fb_Ping();
			fb_TcpOpen();
			fb_TcpServer();
			fb_TcpClient();
			fb_TcpSend();
			fb_TcpRecv();
			fb_TcpClose();
			fb_CfgGetIPAddr();

			TON_TCP_EnDelay.IN 	:= TRUE;
			TON_TCP_EnDelay.PT 	:= t#100ms;
			TON_TCP_EnDelay();
			IF TON_TCP_EnDelay.Q THEN
				TON_TCP_EnDelay(IN := FALSE);
				TCP_Status := INITIAL_PING;
			END_IF

		INITIAL_PING:
			fb_Ping.enable 		:= TRUE;
			fb_Ping.IP_Address 	:= IP_Address;
			fb_Ping();
			IF NOT Enable_Com THEN
				TCP_Status 	:= DISABLED;
			ELSIF fb_Ping.PING_OK THEN
				PING_OK 	:= TRUE;
				IF ETH_Card = '' THEN
					TCP_Status 	:= OPEN_TCP;
				ELSE
					TCP_Status 	:= READ_LOCAL_IP;
				END_IF
			ELSIF fb_Ping.ERROR THEN
				ERR_NO_RESPONSE := fb_Ping.ERR_NO_RESPONSE;
				ERR_INTERNAL	:= fb_Ping.ERR_INTERNAL;
				TCP_Status 		:= RECONNECTION;
			END_IF

		READ_LOCAL_IP:
			fb_CfgGetIPAddr.enable 	:= TRUE;
			fb_CfgGetIPAddr.pDevice := ADR(ETH_Card);
			fb_CfgGetIPAddr.pIPAddr := ADR(IP_AdressLocal);
			fb_CfgGetIPAddr.Len 	:= SIZEOF(IP_AdressLocal);
			fb_CfgGetIPAddr();
			IF fb_CfgGetIPAddr.status = ERR_FUB_BUSY THEN
				readResponse := TRUE;
			END_IF
			IF readResponse THEN
				IF fb_CfgGetIPAddr.status = ERR_OK AND NOT (IP_AdressLocal = 'ERROR') THEN
					IP_LocalValid := TRUE;
					TCP_Status 		:= OPEN_TCP;
				ELSIF fb_CfgGetIPAddr.status <> ERR_FUB_BUSY OR (IP_AdressLocal = 'ERROR') THEN
					IP_LocalValid := FALSE;
					TCP_Status 		:= OPEN_TCP;
				END_IF
			END_IF

		OPEN_TCP:
			fb_TcpOpen.enable	:= TRUE;
			IF IP_LocalValid THEN
				fb_TcpOpen.pIfAddr 	:= ADR(IP_AdressLocal);
			ELSE
				fb_TcpOpen.pIfAddr 	:= 0;
			END_IF
			fb_TcpOpen.port 	:= Local_Port;
			fb_TcpOpen.options 	:= tcpOPT_REUSEADDR;
			fb_TcpOpen();
			IF fb_TcpOpen.status = ERR_FUB_BUSY THEN
				readResponse := TRUE;
			END_IF
			IF readResponse THEN
				IF fb_TcpOpen.status = ERR_OK THEN
					IF Enable_Server THEN
						TCP_Status := CFG_SERVER;
					ELSE
						TCP_Status := CFG_CLIENT;
					END_IF
				ELSIF fb_TcpOpen.status = tcpERR_SOCKET_BIND THEN
					ERR_NO_RESPONSE	:= FALSE;
					TCP_Status 		:= CLOSE2;
				END_IF
			END_IF
			IF NOT Enable_Com THEN
				TCP_Status 	:= CLOSE2;
			END_IF

		CFG_SERVER:
			fb_TcpServer.enable 	:= TRUE;
			fb_TcpServer.ident 		:= fb_TcpOpen.ident;
			fb_TcpServer.backlog 	:= 1;
			fb_TcpServer.pIpAddr 	:= ADR(WhoIsConnected);
			fb_TcpServer();
			TON_ConnectionTimeOut.IN := fb_TcpServer.status = ERR_FUB_BUSY;
			TON_ConnectionTimeOut.PT := t#20s;
			TON_ConnectionTimeOut();
			IF fb_TcpServer.status = ERR_FUB_BUSY THEN
				readResponse := TRUE;
			END_IF
			IF readResponse THEN
				IF fb_TcpServer.status = ERR_OK THEN
					TCP_Status 	:= ESTABLISHED_CONNECTION_AS_SERVER;
				ELSIF (fb_TcpServer.status <> ERR_FUB_BUSY) AND (fb_TcpServer.status <> ERR_OK) THEN
					TCP_Status 		:= CLOSE1;
					ERR_INTERNAL	:= TRUE;
				END_IF
			END_IF
//			IF NOT Enable_Com OR TON_ConnectionTimeOut.Q THEN
//				TCP_Status 	:= CLOSE2;
//			END_IF

		CFG_CLIENT:
			fb_TcpClient.enable 	:= TRUE;
			fb_TcpClient.ident 		:= fb_TcpOpen.ident;
			fb_TcpClient.portserv 	:= Remote_Port;
			fb_TcpClient.pServer 	:= ADR(IP_Address);
			fb_TcpClient();
			IF fb_TcpClient.status = ERR_FUB_BUSY THEN
				readResponse := TRUE;
			END_IF
			IF readResponse THEN
				IF fb_TcpClient.status = ERR_OK THEN
					TCP_Status 	:= ESTABLISHED_CONNECTION_AS_CLIENT;
				ELSIF (fb_TcpClient.status <> ERR_FUB_BUSY) AND (fb_TcpClient.status <> ERR_OK) THEN
					ERR_INTERNAL	:= TRUE;
					TCP_Status 		:= CLOSE1;
				END_IF
			END_IF
			IF NOT Enable_Com THEN
				TCP_Status 	:= CLOSE1;
			END_IF

		ESTABLISHED_CONNECTION_AS_SERVER:
			TON_SendTime.IN := (TCP_CommStatus = RECEIVE_DATA);
			TON_SendTime.PT := Send_Time_Act;
			TON_SendTime();

			CASE TCP_CommStatus OF
				COMM_IDLE:
					TCP_CommStatus	:= SEND_DATA;

				SEND_DATA:
					fb_TcpSend.enable 	:= TRUE;
					fb_TcpSend.ident 	:= fb_TcpServer.identclnt;
					fb_TcpSend.pData 	:= Send_Buffer;
					fb_TcpSend.datalen 	:= Send_Length;
					fb_TcpSend();

					IF fb_TcpSend.status = ERR_FUB_BUSY THEN
						commResponse := TRUE;
					END_IF

					IF commResponse THEN
						IF fb_TcpSend.status	= ERR_OK THEN
							TCP_CommStatus	:= RECEIVE_DATA;
						ELSIF fb_TcpSend.status	= tcpERR_NOT_CONNECTED OR fb_TcpSend.status	= tcpERR_SYSTEM THEN
							TON_RcvTimeOut.IN := TRUE;
						END_IF
					END_IF

					IF TON_RcvTimeOut.Q THEN
						TON_RcvTimeOut.IN	:= FALSE;
						TCP_CommStatus		:= COMM_PING;
					END_IF

				RECEIVE_DATA:
					fb_TcpRecv.enable 	:= TRUE;
					fb_TcpRecv.ident 	:= fb_TcpServer.identclnt;
					fb_TcpRecv.pData 	:= Recv_Buffer;
					fb_TcpRecv.datamax 	:= Recv_Length;
					fb_TcpRecv();

					IF commResponse THEN
						IF TON_SendTime.Q AND (fb_TcpRecv.status = ERR_OK OR fb_TcpRecv.status = tcpERR_NO_DATA) THEN
							TCP_CommStatus	:= SEND_DATA;
						ELSIF fb_TcpRecv.status	= tcpERR_NOT_CONNECTED OR fb_TcpRecv.status	= tcpERR_NO_DATA OR fb_TcpSend.status = tcpERR_SYSTEM THEN
							TON_RcvTimeOut.IN := TRUE;
						ELSIF NOT fb_TcpRecv.status = ERR_FUB_BUSY OR fb_TcpRecv.status = ERR_OK THEN
							TON_RcvTimeOut.IN := FALSE;
						END_IF
					END_IF

					IF fb_TcpRecv.status = ERR_FUB_BUSY THEN
						commResponse := TRUE;
					END_IF

					IF TON_RcvTimeOut.Q THEN
						TON_RcvTimeOut.IN	:= FALSE;
						TCP_CommStatus		:= COMM_PING;
					END_IF

				COMM_PING:
					fb_Ping.enable 		:= TRUE;
					fb_Ping.IP_Address 	:= IP_Address;
					fb_Ping();
					IF fb_Ping.PING_OK THEN
						PING_OK 		:=	TRUE;
						TCP_CommStatus	:= RECEIVE_DATA;
					ELSIF fb_Ping.ERROR THEN
						ERR_NO_RESPONSE := fb_Ping.ERR_NO_RESPONSE;
						ERR_INTERNAL	:= fb_Ping.ERR_INTERNAL;
						TCP_Status 		:= CLOSE1;
					END_IF

			END_CASE

			TON_RcvTimeOut.PT := Rcv_Time_Out;
			TON_RcvTimeOut();

			IF TON_RcvTimeOut.Q OR NOT Enable_Com THEN
				TCP_Status 		:= CLOSE1;
				ERR_NO_RESPONSE := TRUE;
			END_IF

		ESTABLISHED_CONNECTION_AS_CLIENT:
			TON_SendTime.IN := (TCP_CommStatus = RECEIVE_DATA);
			TON_SendTime.PT := Send_Time_Act;
			TON_SendTime();

			CASE TCP_CommStatus OF
				COMM_IDLE:
					TCP_CommStatus	:= SEND_DATA;

				SEND_DATA:
					fb_TcpSend.enable 	:= TRUE;
					fb_TcpSend.ident 	:= fb_TcpOpen.ident;
					fb_TcpSend.pData 	:= Send_Buffer;
					fb_TcpSend.datalen 	:= Send_Length;
					fb_TcpSend();

					IF fb_TcpSend.status = ERR_FUB_BUSY THEN
						commResponse := TRUE;
					END_IF

					IF commResponse THEN
						IF fb_TcpSend.status = ERR_OK THEN
							TCP_CommStatus	:= RECEIVE_DATA;
						ELSIF fb_TcpSend.status	= tcpERR_NOT_CONNECTED OR fb_TcpSend.status	= tcpERR_SYSTEM THEN
							TON_RcvTimeOut.IN := TRUE;
						END_IF
					END_IF

					IF TON_RcvTimeOut.Q THEN
						TON_RcvTimeOut.IN	:= FALSE;
						TCP_CommStatus		:= COMM_PING;
					END_IF

				RECEIVE_DATA:
					fb_TcpRecv.enable 	:= TRUE;
					fb_TcpRecv.ident 	:= fb_TcpOpen.ident;
					fb_TcpRecv.pData 	:= Recv_Buffer;
					fb_TcpRecv.datamax 	:= Recv_Length;
					fb_TcpRecv();

					IF commResponse THEN
						IF TON_SendTime.Q AND (fb_TcpRecv.status = ERR_OK OR fb_TcpRecv.status = tcpERR_NO_DATA) THEN
							TCP_CommStatus	:= SEND_DATA;
						ELSIF fb_TcpRecv.status	= tcpERR_NOT_CONNECTED OR fb_TcpRecv.status	= tcpERR_NO_DATA OR fb_TcpSend.status = tcpERR_SYSTEM THEN
							TON_RcvTimeOut.IN := TRUE;
						ELSIF NOT fb_TcpRecv.status = ERR_FUB_BUSY OR fb_TcpRecv.status = ERR_OK THEN
							TON_RcvTimeOut.IN := FALSE;
						END_IF
					END_IF

					IF fb_TcpRecv.status = ERR_FUB_BUSY THEN
						commResponse := TRUE;
					END_IF

					IF TON_RcvTimeOut.Q THEN
						TON_RcvTimeOut.IN	:= FALSE;
						TCP_CommStatus		:= COMM_PING;
					END_IF

				COMM_PING:
					fb_Ping.enable 		:= TRUE;
					fb_Ping.IP_Address 	:= IP_Address;
					fb_Ping();
					IF fb_Ping.PING_OK THEN
						PING_OK 		:=	TRUE;
						TCP_CommStatus	:= RECEIVE_DATA;
					ELSIF fb_Ping.ERROR THEN
						ERR_NO_RESPONSE := fb_Ping.ERR_NO_RESPONSE;
						ERR_INTERNAL	:= fb_Ping.ERR_INTERNAL;
						TCP_Status 		:= CLOSE1;
					END_IF

			END_CASE

			TON_RcvTimeOut.PT := Rcv_Time_Out;
			TON_RcvTimeOut();

			IF TON_RcvTimeOut.Q OR NOT Enable_Com THEN
				TCP_Status 		:= CLOSE1;
				ERR_NO_RESPONSE := TRUE;
			END_IF

		CLOSE1:
			IF Enable_Server THEN
				PING_OK := FALSE;
				fb_TcpClose.enable 	:= TRUE;
				fb_TcpClose.ident 	:= fb_TcpServer.identclnt;
				fb_TcpClose();
				IF fb_TcpClose.status = ERR_FUB_BUSY THEN
					readResponse := TRUE;
				END_IF
				IF readResponse THEN
					IF fb_TcpClose.status = ERR_OK OR fb_TcpClose.status = tcpERR_INVALID_IDENT THEN
						TCP_Status 	:= CLOSE2;
					END_IF
				END_IF
			ELSE
				TCP_Status 	:= CLOSE2;
			END_IF

		CLOSE2:
			PING_OK := FALSE;
			fb_TcpClose.enable 	:= TRUE;
			fb_TcpClose.ident 	:= fb_TcpOpen.ident;
			fb_TcpClose();
			IF fb_TcpClose.status = ERR_FUB_BUSY THEN
				readResponse := TRUE;
			END_IF
			IF readResponse THEN
				IF fb_TcpClose.status = ERR_OK OR fb_TcpClose.status = tcpERR_INVALID_IDENT THEN
					IF NOT Enable_Com THEN
						TCP_Status 	:= DISABLED;
					ELSE
						TCP_Status 	:= RECONNECTION;
					END_IF
				END_IF
			END_IF

		RECONNECTION:
			PING_OK := FALSE;
			TON_TCP_EnDelay.IN := TRUE;
			IF ConnectionAttempt = 0 THEN
				TON_TCP_EnDelay.PT := t#100ms;
			ELSIF ConnectionAttempt < 5 THEN
				TON_TCP_EnDelay.PT := t#5s;
			ELSIF ConnectionAttempt < 11 THEN
				TON_TCP_EnDelay.PT := t#30s;
			ELSIF ConnectionAttempt < 20 THEN
				TON_TCP_EnDelay.PT := t#5m;
			END_IF
			TON_TCP_EnDelay();
			IF TON_TCP_EnDelay.Q THEN
				TON_TCP_EnDelay(IN := FALSE);
				ConnectionAttempt := ConnectionAttempt + 1;
				TCP_Status := INITIALIZE_FB;
			ELSIF NOT Enable_Com THEN
				TCP_Status 	:= DISABLED;
			END_IF
	END_CASE

	IF TCP_Status <> oldTCP_Status THEN
		oldTCP_Status := TCP_Status;
		TON_ConnectionTimeOut(IN := FALSE);
		readResponse := FALSE;
	END_IF

	IF TCP_CommStatus <> oldTCP_CommStatus THEN
		oldTCP_CommStatus := TCP_CommStatus;
		commResponse := FALSE;
	END_IF

	TON_Connection_OK.IN := (TCP_Status = ESTABLISHED_CONNECTION_AS_SERVER) OR (TCP_Status = ESTABLISHED_CONNECTION_AS_CLIENT);
	TON_Connection_OK.PT := t#3s;
	TON_Connection_OK();
	Connection_OK := TON_Connection_OK.Q;

	IF Connection_OK THEN
		ConnectionAttempt 	:= 0;
		ERR_INTERNAL		:= FALSE;
		ERR_NO_RESPONSE		:= FALSE;
	END_IF

	ERROR := ERR_INTERNAL OR ERR_NO_RESPONSE;
END_FUNCTION_BLOCK
```

#### PING_Fun.st
```iecst
FUNCTION_BLOCK PING_Fun
	IF NOT enable THEN
		PING_OK 			:= FALSE;
		ERR_NO_RESPONSE 	:= FALSE;
		ERR_INTERNAL	 	:= FALSE;
		ERROR 				:= FALSE;
		Status 				:= NO_EXECUTION;
		RETURN;
	END_IF;
	Fb_IcmpPing.pHost	:= ADR(IP_Address);
	Fb_IcmpPing.timeout := 50;
	CASE Status OF
		NO_EXECUTION:
			Fb_IcmpPing.enable  := FALSE;
			readResponse 	:= FALSE;
			PachetSent		:= 0;
			PachetRecived	:= 0;
			PachetLoss		:= 0;
			IF enable THEN
				Status := EXECUTION;
			END_IF;

		EXECUTION:
			Fb_IcmpPing.enable  := TRUE;
			IF Fb_IcmpPing.status = ERR_FUB_BUSY THEN
				readResponse := TRUE;
			END_IF
			IF readResponse THEN
				CASE Fb_IcmpPing.status OF
					ERR_OK:
						PachetSent 		:= PachetSent +1;
						PachetRecived 	:= PachetRecived +1;

					icmpERR_NO_RESPONSE:
						PachetSent 		:= PachetSent +1;
						PachetLoss 		:= PachetLoss +1;

					ERR_FUB_BUSY,
					ERR_FUB_ENABLE_FALSE:

					icmpERR_PARAMETER,
					icmpERR_SOCKET_CREATE,
					icmpERR_SYSTEM:
						Status := ERROR_INTERNAL;
				END_CASE;
			END_IF
			IF PachetSent >= 4 THEN
				IF PachetLoss >= 1 THEN
					Status := NO_RESPONSE;
				ELSE
					Status := SUCCESSFUL;
				END_IF
			END_IF

		SUCCESSFUL, NO_RESPONSE, ERROR_INTERNAL:
			Fb_IcmpPing.enable  := FALSE;

	END_CASE;
	Fb_IcmpPing();

	PING_OK 			:= Status = SUCCESSFUL;
	ERR_NO_RESPONSE 	:= Status = NO_RESPONSE;
	ERR_INTERNAL	 	:= Status = ERROR_INTERNAL;
	ERROR 				:= ERR_NO_RESPONSE OR ERR_INTERNAL;
END_FUNCTION_BLOCK
```

### Library Logical/00_AID/Libraries/Sidel_Libraries/ITC/UDP_COM (IEC, version 3.00.0)

#### UDP_COM.typ - UDP Communication Type
```iecst
(********************************************************************
 * COPYRIGHT - Sidel Spa
 ********************************************************************
 * Library: UDP_COM
 * File: UDP_COM.typ
 * Author: Andrea.Cortesi
 * Created: May 28, 2013
 ********************************************************************
 * Data types of library UDP_COM
 ********************************************************************)

TYPE
	UDP_DataType : 	STRUCT
		Connection_OK : BOOL;
		Com_Status : UINT; (*(0=Connect OK;1=Not Enabled;2=Error Sending;3=Error Receiving;10=Connection Waiting)*)
	END_STRUCT;
END_TYPE
```

#### UDP_COM.var - UDP Communication Var
```iecst
(********************************************************************
 * COPYRIGHT -- Sidel
 ********************************************************************
 * Library: UDP_COM
 * File: UDP_COM.var
 * Author: Andrea.Cortesi
 * Created: May 28, 2013
 ********************************************************************
 * Constants of library UDP_COM
 ********************************************************************)
VAR CONSTANT
	UDP_Connected_OK : USINT := 0;
	UDP_Not_Enabled : USINT := 1;
	UDP_Error_Sending : USINT := 2;
	UDP_Error_Receiving : USINT := 3;
	UDP_Connection_Close : USINT := 4;
	UDP_Connection_Waiting : USINT := 10;
END_VAR
```

#### UDP_COM.fun - UDP Exported functions and function blocks
```iecst
(********************************************************************
 * COPYRIGHT -- Sidel
 ********************************************************************
 * Library: UDP_COM
 * File: UDP_COM.fun
 * Author: Andrea.Cortesi
 * Created: May 28, 2013
 ********************************************************************
 * Functions and function blocks of library UDP_COM
 ********************************************************************)

FUNCTION_BLOCK UDP_COM (*UDP Communication Function*)
	VAR_INPUT
		Enable_Com : BOOL; (*Enable Communication*)
		IP_Address : STRING[40]; (*Partner IP address. (e.g. '10.1.92.20') (as a string)*)
		Local_Port : UINT; (*Local port number.*)
		Remote_Port : UINT; (*Remote port number.*)
		Recv_Buffer : UDINT; (*Received data buffer address (string given as a pointer)*)
		Recv_Length : UDINT; (*Reiceved data maximum length (in bytes)*)
		Send_Buffer : UDINT; (*Data to send buffer address (string given as a pointer)*)
		Send_Length : UDINT; (*Sent data length (in bytes)*)
		Rcv_Time_Out : TIME; (*Reception time out setpoint (in ms) (typical value: 1000ms)*)
		Send_Time_Act : TIME; (*Data send time cadence (in ms) (typical value: 100ms)*)
	END_VAR
	VAR_OUTPUT
		Connection_OK : BOOL; (*True = both PLCs are connected*)
		Recv_Data_Length : UDINT; (*Length of the bytes received.*)
		Send_Data_Length : UDINT; (*Length of the bytes send*)
		Status : USINT; (*Communication status. Status = 0, means communication is OK*)
		Status_Message : STRING[25]; (*Communication status string*)
	END_VAR
	VAR
		Socket_ID : UDINT; (*Identifier sent by the UdpOpen block *)
		UDP_Com_UdpOpen : UdpOpen; (*Communication opening function block*)
		UDP_Com_UdpClose : UdpClose; (*Communication closing function block*)
		UDP_Com_UdpSend : UdpSend; (*Data sending function block*)
		UDP_Com_UdpRecv : UdpRecv; (*Data receiving function block*)
		UDP_Step : USINT; (*Implemented communication block status*)
		Open_Status : UINT; (*Communication opening function block status*)
		Send_Status : UINT; (*Data sending function block status*)
		Recv_Status : UINT; (*Data receiving function block status*)
		Close_Status : UINT; (*communication closing function block status*)
		Send_Timer : TON; (*Sending timer*)
		Rcv_Timer : TON; (*Receiveing timer*)
		ConnectTimeOut_Timer : TON; (*Connection Time Out*)
	END_VAR
END_FUNCTION_BLOCK
```

#### UDP_COM.st - UDP Communication St
```iecst
(********************************************************************
 * COPYRIGHT -- Sidel
 ********************************************************************
 * Library: UDP_COM
 * File: UDP_COM.st
 * Author: Andrea.Cortesi
 * Created: Jun 26, 2013
 ********************************************************************
 * Implementation of library UDP_COM
 ********************************************************************)

(* UDP COMMUNICATION FUNCTION BLOC IMPLEMENTATION *)
FUNCTION_BLOCK UDP_COM

	Send_Timer.PT := Send_Time_Act;
	Send_Timer();

	Rcv_Timer.PT := Rcv_Time_Out;
	Rcv_Timer();

	ConnectTimeOut_Timer.PT := T#2000ms;
	ConnectTimeOut_Timer();

	IF Rcv_Timer.Q THEN
		(* Close Communication UDP *)
		UDP_Step := 60;
	END_IF

	CASE UDP_Step OF

		0:	(* Open UDP Connection *)

			Rcv_Timer.IN := FALSE;

			IF Enable_Com THEN
				Status := UDP_Connection_Waiting;
			ELSE
				Status := UDP_Not_Enabled;
			END_IF

			UDP_Com_UdpOpen.enable	 := Enable_Com;
			UDP_Com_UdpOpen.pIfAddr  := 0;           (* Listen on all UDP Interfaces*)
			UDP_Com_UdpOpen.port 	 := Local_Port;  (* Port to listen*)
			UDP_Com_UdpOpen.options  := udpOPT_REUSEADDR;

			UDP_Com_UdpOpen();    (* Call the Function*)

			Socket_ID 	             := UDP_Com_UdpOpen.ident;
			Open_Status              := UDP_Com_UdpOpen.status;

			IF Open_Status = 0 THEN  (* UdpOpen successful*)
				(* Initialization Send and Receive Ident *)
				UDP_Step := 40;
			END_IF

			Connection_OK := FALSE;

		40: (* Initialization Send and Receive Ident *)

			Rcv_Timer.IN := TRUE;

			(* Data send block parameters *)
			UDP_Com_UdpSend.enable  := TRUE;
			UDP_Com_UdpSend.ident   := Socket_ID;	                    (* Client Ident from UDP_Open *)
			UDP_Com_UdpSend.pHost   := ADR(IP_Address);	                (* IP Address of remote partner *)
			UDP_Com_UdpSend.port    := Remote_Port;		                (* Port number of remote partner *)
			UDP_Com_UdpSend.pData   := Send_Buffer;	                    (* Which data to send *)
			UDP_Com_UdpSend.datalen := Send_Length;	                    (* Lenght of data to send *)
			UDP_Com_UdpSend.flags   := 0;

			(* Data receive block parameters *)
			UDP_Com_UdpRecv.enable  := TRUE;
			UDP_Com_UdpRecv.ident   := Socket_ID;	                    (* Client Ident from UDP_Open *)
			UDP_Com_UdpRecv.pIpAddr := ADR(IP_Address);	                (* IP Address of remote partner *)
			UDP_Com_UdpRecv.pData   := Recv_Buffer;	                    (* Where to store the incoming data *)
			UDP_Com_UdpRecv.datamax := Recv_Length;                     (* Lenght of data buffer *)
			UDP_Com_UdpRecv.flags   := 0;

			UDP_Step := 50;

			IF NOT(Enable_Com) THEN
				UDP_Step := 0;
			END_IF

			Connection_OK := FALSE;

		50: (* Send and Receive Data *)

			Send_Timer.IN := NOT(Send_Timer.Q);

			UDP_Com_UdpRecv();  (* Call the "Data Recv" function block *)

			Recv_Status        := UDP_Com_UdpRecv.status;
			Recv_Data_Length   := UDP_Com_UdpRecv.recvlen;

			IF Send_Timer.Q THEN
				UDP_Com_UdpSend.enable := TRUE;
			END_IF

			UDP_Com_UdpSend();	(* Call the "Data Sent" function block *)

			Send_Status        := UDP_Com_UdpSend.status;
			Send_Data_Length   := UDP_Com_UdpSend.sentlen;
			Status 	 	       := UDP_Connected_OK;

			IF UDP_Com_UdpSend.enable THEN

				IF (Send_Status <> 65535) AND (Send_Status <> 0) THEN
					UDP_Step := 60;
					Status   := UDP_Error_Sending;
				END_IF

				IF (Send_Status = 0) THEN
					Send_Timer.IN := FALSE;
				ELSE
					Send_Timer.IN := TRUE;
				END_IF

			END_IF

			IF (Recv_Status <> 65535) AND (Recv_Status <> 0) AND (Recv_Status <> udpERR_NO_DATA) THEN
				UDP_Step := 60;
				Status   := UDP_Error_Receiving;
			END_IF

			IF (Recv_Status = 0) THEN
				Rcv_Timer.IN := FALSE;
			ELSE
				Rcv_Timer.IN := TRUE;
			END_IF

			IF NOT(Enable_Com) THEN
				UDP_Step := 60;
			END_IF

			Connection_OK := TRUE;

		60: (* Close Communication UDP *)

			Rcv_Timer.IN := FALSE;

			UDP_Com_UdpClose.enable := TRUE;
			UDP_Com_UdpClose.ident  := Socket_ID;
			UDP_Com_UdpClose();

			Close_Status := UDP_Com_UdpClose.status;
			Status 	 	 := UDP_Connection_Close;

			IF (Close_Status = 0) THEN
				UDP_Step := 70;
			END_IF

			Connection_OK := FALSE;

		70: (* Wait Open New Connection *)

			Rcv_Timer.IN            := FALSE;
			ConnectTimeOut_Timer.IN := TRUE;

			IF ConnectTimeOut_Timer.Q THEN
				UDP_Step                := 0;
				ConnectTimeOut_Timer.IN := FALSE;
			END_IF

			Status 	 	  := UDP_Connection_Waiting;
			Connection_OK := FALSE;

		ELSE

			UDP_Step := 60;

	END_CASE

	CASE Status OF

		0: Status_Message := 'UDP Connection OK';
		1: Status_Message := 'UDP Not Enabled';
		2: Status_Message := 'UDP Error Sending';
		3: Status_Message := 'UDP Error Receiving';
		4: Status_Message := 'UDP Connection Close';
		5: Status_Message := 'UDP Send Receive Run';
	   10: Status_Message := 'UDP Connection Waiting';

	ELSE
		   Status_Message := 'Not Define';
	END_CASE

END_FUNCTION_BLOCK
```

### Library Logical/00_AID/Libraries/Sidel_Libraries/ITC/ETHIP_COM (IEC, version 4.00.1) - 4.00.1 - ETHIP COM Library by Sidel
Depends on: AsEthIP, AsICMP, AsString, Runtime, Standard

#### ETHIP_COM.typ - ETHIP COM Data Types
```iecst
TYPE
	ETHIP_Status_Type :
		(
		ETHIP_DISABLED,
		ETHIP_INITIALIZE_FB,
		ETHIP_INITIAL_PING,
		ETHIP_OPEN,
		ETHIP_RUNNING,
		ETHIP_CLOSE,
		ETHIP_PING,
		ETHIP_WAIT_RESET,
		ETHIP_RECONNECTION
		);
END_TYPE
```

#### ETHIP_COM.var - ETHIP COM Constants
```iecst
(********************************************************************
 * COPYRIGHT --  Sidel S.p.a
 ********************************************************************
 * Library: ETHIP_COM
 * File: ETHIP_COM.var
 * Author: Andrea.Cortesi
 * Created: August 26, 2015
 ********************************************************************
 * Constants of library ETHIP_COM
 ********************************************************************)
VAR CONSTANT
	Buffer_Status_MaxLimit : USINT := 40;
END_VAR
```

#### ETHIP_COM.fun - ETHIP COM Functions and Function Blocks
```iecst
(********************************************************************
 * COPYRIGHT --  Sidel S.p.a.
 ********************************************************************
 * Library: ETHIP_COM
 * File: ETHIP_COM.fun
 * Author: Andrea.Cortesi
 * Created: August 26, 2015
 ********************************************************************
 * Functions and function blocks of library ETHIP_COM
 ********************************************************************)

FUNCTION_BLOCK ETHIP_COM
	VAR_INPUT
		Enable : BOOL := FALSE; (*Enable Function Block*)
		IP_Address_Partner : STRING[16] := ' '; (*IP Address Partner*)
		Alive_Bit_From_Partner : BOOL := FALSE; (*Alive Bit From Partner*)
		Reset : BOOL := FALSE; (*Reset Button*)
		TimeOut_Value : UINT := 5000; (*(OPTIONAL) TimeOut Value [ms]. Default value if no setting is 5000 [ms]. Min value accepted 3000 [ms]*)
		Config_DataObject : UDINT := 0; (*Pointer to Data Object Configuration*)
	END_VAR
	VAR_OUTPUT
		Error : BOOL := FALSE; (*Error: TimeOut Connnection or Internal Error (ex: Data Object Not correct) or other function error*)
	END_VAR
	VAR
		PING_Partner : IcmpPing := (0);
		ConnectionAttempt : UINT;
		ETHIP_Init : EIPInit := (0);
		ETHIP_Cyclic : EIPCyclic := (0);
		ETHIP_Exit : EIPExit := (0);
		Handle_Init : UDINT := 0;
		Status : UINT := 0;
		Status_Old : UINT := 0;
		Step_Msg_Active : STRING[255] := ' ';
		Step_Msg_Active_Old : STRING[255] := ' ';
		Msg_Error : STRING[255] := ' ';
		Status_String : STRING[255] := ' ';
		Buffer_Status : ARRAY[0..Buffer_Status_MaxLimit] OF STRING[255] := [41(' ')]; (*Buffer Diagnostic for Status Message*)
		Buffer_Status_Index : USINT := 0;
		Timer_StartComDelay : TON := (0);
		Timer_CommTimeOut : TON := (0);
		Error_Internal : BOOL := FALSE;
		Ping_Ok : BOOL := FALSE;
		ComInit : BOOL := FALSE;
		ComStart : BOOL := FALSE;
		ComExit : BOOL := FALSE;
		zzEdge00000 : BOOL;
		zzEdge00001 : BOOL;
		zzEdge00002 : BOOL;
		zzEdge00003 : BOOL;
	END_VAR
END_FUNCTION_BLOCK
```
